(* IEC 61131-3 sources: inproshop/test9_exported/1.Function/FB/Socket(套接字), 6 files *)

(* ---- Str_TcpClient.st ---- *)
TYPE Str_TcpClient :
STRUCT
	Enable:		BOOL;//使能
	Execute:	BOOL;//发送数据
	SrcTcpPort:	UINT;//本地端口号
	DstAdr:		STRING;//远程IP地址
	DstTcpPort:	UINT;//远程端口号
	SendDat:	ARRAY[0..500] OF BYTE;//发送数据内容
	SendSize:	UINT;//发送数据长度
	RcvDat:		ARRAY[0..500] OF BYTE;//接收数据内容
	RcvSize:	UINT;//接收数据长度
	Active:		BOOL;//	链接已建立
	SendDone:	BOOL;//	发送数据完成
	RcvDone:	BOOL;//	接收数据完成
	Error:		BOOL;//	错误
	ErrorID:	WORD;//	错误代码
END_STRUCT
END_TYPE

(* ---- Str_TcpClient_String.st ---- *)
TYPE Str_TcpClient_String :
STRUCT
	Enable:		BOOL;//使能
	Execute:	BOOL;//发送数据
	SrcTcpPort:	UINT;//本地端口号
	DstAdr:		STRING;//远程IP地址
	DstTcpPort:	UINT;//远程端口号
	SendDat:	STRING(500);//发送数据内容
	RcvDat:		STRING(500);//接收数据内容
	Active:		BOOL;//	链接已建立
	SendDone:	BOOL;//	发送数据完成
	RcvDone:	BOOL;//	接收数据完成
	Error:		BOOL;//	错误
	ErrorID:	WORD;//	错误代码
END_STRUCT
END_TYPE

(* ---- Str_TcpClient_Wstring.st ---- *)
TYPE Str_TcpClient_Wstring :
STRUCT
	Enable:		BOOL;//使能
	Execute:	BOOL;//发送数据
	SrcTcpPort:	UINT;//本地端口号
	DstAdr:		STRING[256];//远程IP地址
	DstTcpPort:	UINT;//远程端口号
	SendDat:	WSTRING(500);//发送数据内容
	RcvDat:		WSTRING(500);//接收数据内容
	Active:		BOOL;//	链接已建立
	SendDone:	BOOL;//	发送数据完成
	RcvDone:	BOOL;//	接收数据完成
	Error:		BOOL;//	错误
	ErrorID:	WORD;//	错误代码
END_STRUCT
END_TYPE

(* ---- FB_TcpClient.st ---- *)
FUNCTION_BLOCK FB_TcpClient
VAR_IN_OUT
	ioTcpClient:Str_TcpClient;
END_VAR
VAR_OUTPUT
END_VAR
VAR
	i:UINT;//循环变量
	STR1:POINTER TO STRING(500);
	STR2:POINTER TO STRING(500);
	LEN_Rcv:ULINT;
	RcvDat:ARRAY[0..500] OF BYTE;

END_VAR
VAR
	TCP_Client_instance: TCP_Client;
	TCP_Send_instance: TCP_Send;
	TCP_Receive_instance: TCP_Receive;
END_VAR

TCP_Client_instance(
	xEnable:= ioTcpClient.Enable,
	strIpAddrDst:= ioTcpClient.DstAdr,
	uiPortDst:= ioTcpClient.DstTcpPort,
	udiTimeOut:= ,
	xNotKeepAlive:= ,
	xDone=> ,
	xBusy=> ,
	xError=> ,
	dwErrorID=> ,
	xActive=> ioTcpClient.Active,
	hConnection=> );

TCP_Send_instance(
	xExecute:= ioTcpClient.Execute AND TCP_Client_instance.xActive,
	hConnection:= TCP_Client_instance.hConnection,
	uiSize:=ioTcpClient.SendSize,
	pbyData:= ADR(ioTcpClient.SendDat),
	udiTimeOut:= ,
	xDone=> ,
	xBusy=> ,
	xError=> ,
	dwErrorID=> );

TCP_Receive_instance(
	xEnable:= TCP_Client_instance.xActive AND NOT TCP_Receive_instance.xDone AND NOT TCP_Receive_instance.xError,
	hConnection:= TCP_Client_instance.hConnection,
	uiSize:= 500,
	pbyData:= ADR(RcvDat),
	xDone=> ,
	xBusy=> ,
	xError=> ,
	dwErrorID=> ,
	xReady=> ,
	uiCount=> LEN_Rcv);

//截取字符串长度
IF LEN_Rcv<> 0 THEN
	FOR i:=0 TO 500 BY 1 DO
		ioTcpClient.RcvDat[i]:=0;
	END_FOR
	FOR i:=0 TO ULINT_TO_UINT(LEN_Rcv) BY 1 DO
		ioTcpClient.RcvDat[i]:=RcvDat[i];
	END_FOR
	ioTcpClient.RcvDone:=TRUE;
	ioTcpClient.RcvSize:=ULINT_TO_UINT(LEN_Rcv);
ELSE
	ioTcpClient.RcvDone:=FALSE;
END_IF

//发送指令OFF
IF TCP_Send_instance.xDone OR TCP_Send_instance.xError OR NOT ioTcpClient.Enable THEN
	ioTcpClient.Execute:=FALSE;
END_IF

(* ---- FB_TcpClient_String.st ---- *)
FUNCTION_BLOCK FB_TcpClient_String
VAR_IN_OUT
	ioTcpClient:Str_TcpClient_String;
END_VAR
VAR_OUTPUT
END_VAR
VAR
	i:UINT;//循环变量
	STR1:POINTER TO STRING(500);
	STR2:POINTER TO STRING(500);
	LEN_Rcv:ULINT;
	RcvDat:STRING(500);

END_VAR
VAR
	TCP_Client_instance: TCP_Client;
	TCP_Send_instance: TCP_Send;
	TCP_Receive_instance: TCP_Receive;
END_VAR

TCP_Client_instance(
	xEnable:= ioTcpClient.Enable,
	strIpAddrDst:= ioTcpClient.DstAdr,
	uiPortDst:= ioTcpClient.DstTcpPort,
	udiTimeOut:= ,
	xNotKeepAlive:= ,
	xDone=> ,
	xBusy=> ,
	xError=> ,
	dwErrorID=> ,
	xActive=> ioTcpClient.Active,
	hConnection=> );

TCP_Send_instance(
	xExecute:= ioTcpClient.Execute AND TCP_Client_instance.xActive,
	hConnection:= TCP_Client_instance.hConnection,
	uiSize:=INT_TO_UINT(len(ioTcpClient.SendDat)),
	pbyData:= ADR(ioTcpClient.SendDat),
	udiTimeOut:= ,
	xDone=> ,
	xBusy=> ,
	xError=> ,
	dwErrorID=> );

TCP_Receive_instance(
	xEnable:= TCP_Client_instance.xActive AND NOT TCP_Receive_instance.xDone AND NOT TCP_Receive_instance.xError,
	hConnection:= TCP_Client_instance.hConnection,
	uiSize:= 500,
	pbyData:= ADR(RcvDat),
	xDone=> ,
	xBusy=> ,
	xError=> ,
	dwErrorID=> ,
	xReady=> ,
	uiCount=> LEN_Rcv);

//截取字符串长度
IF LEN_Rcv<> 0 THEN
	FOR i:=0 TO ULINT_TO_UINT(LEN_Rcv) BY 1 DO
		STR2:=ADR(RcvDat)+ULINT_TO_DWORD( LEN_Rcv)+i;
		STR2^:='';
	END_FOR
	ioTcpClient.RcvDone:=TRUE;
ELSE
	ioTcpClient.RcvDone:=FALSE;
END_IF
IF ioTcpClient.RcvDone THEN
	ioTcpClient.RcvDat:=RcvDat;
END_IF

//发送指令OFF
IF TCP_Send_instance.xDone OR TCP_Send_instance.xError OR NOT ioTcpClient.Enable THEN
	ioTcpClient.Execute:=FALSE;
END_IF

(* ---- FB_TcpClient_Wstring.st ---- *)
FUNCTION_BLOCK FB_TcpClient_Wstring
VAR_IN_OUT
	ioTcpClient:Str_TcpClient_Wstring;
END_VAR
VAR_OUTPUT
END_VAR
VAR
	i:UINT;//循环变量
	STR1:POINTER TO WSTRING(500);
	STR2:POINTER TO WSTRING(500);
	LEN_Rcv:ULINT;
	RcvDat:WSTRING(500);

END_VAR
VAR
	TCP_Client_instance: TCP_Client;
	TCP_Send_instance: TCP_Send;
	TCP_Receive_instance: TCP_Receive;
END_VAR

//计算发送字符长度
STR1:=ADR(ioTcpClient.SendDat);
FOR i:= 0 TO 500 BY 2 DO
	STR2:= STR1+UINT_TO_DWORD(i);
	IF STR2^="" THEN
		TCP_Send_instance.uiSize:=i;//获取字符串长度
		EXIT;
	END_IF
END_FOR

TCP_Client_instance(
	xEnable:= ioTcpClient.Enable,
	strIpAddrDst:= ioTcpClient.DstAdr,
	uiPortDst:= ioTcpClient.DstTcpPort,
	udiTimeOut:= ,
	xNotKeepAlive:= ,
	xDone=> ,
	xBusy=> ,
	xError=> ,
	dwErrorID=> ,
	xActive=> ioTcpClient.Active,
	hConnection=> );

TCP_Send_instance(
	xExecute:= ioTcpClient.Execute AND TCP_Client_instance.xActive,
	hConnection:= TCP_Client_instance.hConnection,
	uiSize:= ,
	pbyData:= ADR(ioTcpClient.SendDat),
	udiTimeOut:= ,
	xDone=> ,
	xBusy=> ,
	xError=> ,
	dwErrorID=> );

TCP_Receive_instance(
	xEnable:= TCP_Client_instance.xActive AND NOT TCP_Receive_instance.xDone AND NOT TCP_Receive_instance.xError,
	hConnection:= TCP_Client_instance.hConnection,
	uiSize:= 500,
	pbyData:= ADR(RcvDat),
	xDone=> ,
	xBusy=> ,
	xError=> ,
	dwErrorID=> ,
	xReady=> ,
	uiCount=> LEN_Rcv);

//截取字符串长度
IF LEN_Rcv<> 0 THEN
	FOR i:=0 TO ULINT_TO_UINT(LEN_Rcv) BY 2 DO
		STR2:=ADR(RcvDat)+ULINT_TO_DWORD( LEN_Rcv)+i;
		STR2^:="";
	END_FOR
	ioTcpClient.RcvDone:=TRUE;
ELSE
	ioTcpClient.RcvDone:=FALSE;
END_IF
IF ioTcpClient.RcvDone THEN
	ioTcpClient.RcvDat:=RcvDat;
END_IF

//发送指令OFF
IF TCP_Send_instance.xDone OR TCP_Send_instance.xError OR NOT ioTcpClient.Enable THEN
	ioTcpClient.Execute:=FALSE;
END_IF
